// TIA Portal V18 export
FUNCTION "mixing ratio & material Data" : Void   // FC37, LAD
{ S7_Optimized_Access := 'TRUE' }
VERSION : 0.1
// stored: AutoNumber true, IsIECCheckEnabled false, SetENOAutomatically false, UDAEnableTagReadback false
BEGIN

REGION Network 1 (SCL)
   "Material Data current pgm"."name A+B" := CONCAT(IN1 := "Material Data current pgm".Name.A, IN2 :="Material Data current pgm"."+symbol", IN3 := "Material Data current pgm".Name.B);
END_REGION

REGION Network 2: mixing Ratio according to density
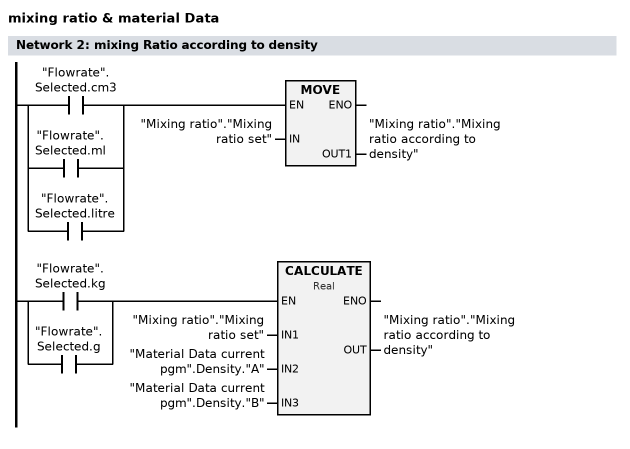
   RUNG wire#powerrail
      Contact( "Flowrate".Selected.cm3 )
      wire#w1
      Move(in := "Mixing ratio"."Mixing ratio set", out1 => "Mixing ratio"."Mixing ratio according to density")
   END_RUNG
   RUNG wire#powerrail
      Contact( "Flowrate".Selected.ml )
   END_RUNG wire#w1
   RUNG wire#powerrail
      Contact( "Flowrate".Selected.litre )
   END_RUNG wire#w1
   RUNG wire#powerrail
      Contact( "Flowrate".Selected.kg )
      wire#w2
      { S7_Templates := "SrcType := Real"; S7_Expression := "(IN1/IN2)*IN3" } Calculate(in1 := "Mixing ratio"."Mixing ratio set", in2 := "Material Data current pgm".Density."A", in3 := "Material Data current pgm".Density."B", out => "Mixing ratio"."Mixing ratio according to density")
   END_RUNG
   RUNG wire#powerrail
      Contact( "Flowrate".Selected.g )
   END_RUNG wire#w2
   // the same network as SCL:
   IF "Flowrate".Selected.cm3 OR "Flowrate".Selected.ml OR "Flowrate".Selected.litre THEN
       "Mixing ratio"."Mixing ratio according to density" := "Mixing ratio"."Mixing ratio set";
   END_IF;
   IF "Flowrate".Selected.kg OR "Flowrate".Selected.g THEN
       "Mixing ratio"."Mixing ratio according to density" := ("Mixing ratio"."Mixing ratio set"/"Material Data current pgm".Density."A")*"Material Data current pgm".Density."B";
   END_IF;
END_REGION
END_FUNCTION
